// TwinCAT 3 PLC project MC
// ProgramVersion: 3.1.4023.0
// libraries:
//   Tc2_EtherCAT, * (Beckhoff Automation GmbH)
//   Tc2_MC2, * (Beckhoff Automation GmbH)
//   Tc2_MC2_Camming, * (Beckhoff Automation GmbH)
//   Tc2_Standard, * (Beckhoff Automation GmbH)
//   Tc2_System, * (Beckhoff Automation GmbH)
//   Tc3_Module, * (Beckhoff Automation GmbH)
// project tree:
//   / GlobalTextList.TcGTLO, PlcTask.TcTTO, 视图管理器.TcVMO (not stored)
//   POUs/ MAIN.TcPOU, Motion01.TcPOU, Test_SDO.TcPOU
//   VISUs/ hmi.TcVIS
// real-time tasks:
//   TASK PlcTask: cycle T#10ms, priority 20, ADS port 350
//   TASK PlcTask1: cycle T#10ms, priority 21, ADS port 351
// motion (NC):
//   TASK NC-Task 1 SAF: cycle T#2ms, priority 4, ADS port 501
//   TASK NC-Task 1 SVB: cycle T#10ms, priority 8, ADS port 511
//   AXIS Axis 1 (id 1)
//     Dynamic: AccelerationMaximum=30000, DecelerationMaximum=30000, Acceleration=10000, Deceleration=10000, Jerk=5000
//     Velo: Maximum=3300
//     OtherSettings: AllowMotionCmdToSlave=true
//     encoder EncType=1
//       EncPara: ScaleFactorNumerator=60, ScaleFactorDenominator=131072
//         Inc: RefSoftSyncMask=#x0001ffff
//     drive DrvType=5
//       Analog: VeloReferenz=3300, TorqueSetpointScale=10, ScaleFactorActTorque=0.1
//       TimeComp: TaskDelayCycles=1
//     controller CtrType=1
//       CtrPara: PriorControlFactor=1
//         PosDiffControl: Range=100
//         Observer: BandWidth=20
//   AXIS Axis 2 (id 2)
//     OtherSettings: AllowMotionCmdToSlave=true
//     encoder EncType=1
//       EncPara: ScaleFactorNumerator=60, ScaleFactorDenominator=131072
//         Inc: RefSoftSyncMask=#x0001ffff
//     drive DrvType=5
//       Analog: TorqueSetpointScale=10, ScaleFactorActTorque=0.1
//       TimeComp: TaskDelayCycles=1
//     controller CtrType=1
//       CtrPara: PriorControlFactor=1
//         PosDiffControl: Range=100
//         Observer: BandWidth=20
//   AXIS master (id 3)
//     OtherSettings: AllowMotionCmdToSlave=true
//     encoder EncType=19
//       EncPara: ScaleFactorNumerator=60, ScaleFactorDenominator=131072, MaxCount=#xffffffff
//         Inc: RefSoftSyncMask=#x0001ffff
//     drive DrvType=16
//       DrvPara: MaxCount=#xffffffff, DriveControlDWord=#x00020100
//         Analog: TorqueSetpointScale=10, ScaleFactorActTorque=0.1
//         TimeComp: TaskDelayCycles=1
//     controller CtrType=1
//       CtrPara: PriorControlFactor=1
//         PosDiffControl: Range=100
//         Observer: BandWidth=20
//   AXIS slave (id 4)
//     OtherSettings: AllowMotionCmdToSlave=true
//     encoder EncType=19
//       EncPara: ScaleFactorNumerator=60, ScaleFactorDenominator=131072, MaxCount=#xffffffff
//         Inc: RefSoftSyncMask=#x0001ffff
//     drive DrvType=16
//       DrvPara: MaxCount=#xffffffff, DriveControlDWord=#x00020000
//         Analog: TorqueSetpointScale=10, ScaleFactorActTorque=0.1
//         TimeComp: TaskDelayCycles=1
//     controller CtrType=1
//       CtrPara: PriorControlFactor=1
//         PosDiffControl: Range=100
//         Observer: BandWidth=20
// I/O:
//   DEVICE Device 1 (EtherCAT), AmsNetId 5.112.215.215.2.1
//     Term 1 (EK1200) [EK1200-5000 EtherCAT Power supply (2A E-Bus)]
//       Term 2 (EK1110) [EK1110 EtherCAT extension]
//     Drive 3 (ID600E CoE Drive) [ID600E EtherCAT(CoE) Drive]
//     Drive 4 (ID600E CoE Drive) [ID600E EtherCAT(CoE) Drive]
// variable links:
//   NC-Task 1 SAF/Axes/master <-> Device 1 (EtherCAT)/Drive 3 (ID600E CoE Drive)
//     Drive/Inputs/In/nDataIn1 <-> 1st Transmit PDO mapping/Following Error Actual Value
//     Drive/Inputs/In/nDataIn3[0] <-> 1st Transmit PDO mapping/Torque Actual Value
//     Drive/Inputs/In/nDcOutputTime <-> InfoData/DcOutputShift
//     Drive/Inputs/In/nState1 <-> 1st Transmit PDO mapping/Statusword
//     Drive/Inputs/In/nState2 <-> 1st Transmit PDO mapping/Statusword @bit 8
//     Drive/Inputs/In/nState4 @bit 1 <-> WcState/InputToggle
//     Drive/Inputs/In/nState4 <-> WcState/WcState
//     Drive/Inputs/In/nState5 <-> 1st Transmit PDO mapping/Mode of Operation Display
//     Drive/Outputs/Out/nCtrl1 <-> 1st Receive PDO mapping/Controlword
//     Drive/Outputs/Out/nCtrl2 <-> 1st Receive PDO mapping/Controlword @bit 8
//     Drive/Outputs/Out/nCtrl5 <-> 1st Receive PDO mapping/Mode of Operation
//     Drive/Outputs/Out/nDataOut1 <-> 1st Receive PDO mapping/Target Position
//     Drive/Outputs/Out/nDataOut2 <-> 1st Receive PDO mapping/Target Velocity
//     Drive/Outputs/Out/nDataOut4[0] <-> 1st Receive PDO mapping/Target Torque
//     Enc/Inputs/In/nDataIn1 <-> 1st Transmit PDO mapping/Position Actual Value
//     Enc/Inputs/In/nDataIn3 <-> 1st Transmit PDO mapping/Touch Probe 1 Positive Edge Position Value
//     Enc/Inputs/In/nDcInputTime <-> InfoData/DcInputShift
//     Enc/Inputs/In/nState4 @bit 1 <-> WcState/InputToggle
//     Enc/Inputs/In/nState4 <-> WcState/WcState
//     Enc/Outputs/Out/nCtrl5 <-> 1st Receive PDO mapping/Touch Probe Function
//     Enc/Outputs/Out/nCtrl6 <-> 1st Receive PDO mapping/Touch Probe Function @bit 8
//   NC-Task 1 SAF/Axes/slave <-> Device 1 (EtherCAT)/Drive 4 (ID600E CoE Drive)
//     Drive/Inputs/In/nDcOutputTime <-> InfoData/DcOutputShift
//     Drive/Inputs/In/nState1 <-> 2nd Transmit PDO mapping/Statusword
//     Drive/Inputs/In/nState2 <-> 2nd Transmit PDO mapping/Statusword @bit 8
//     Drive/Inputs/In/nState4 @bit 1 <-> WcState/InputToggle
//     Drive/Inputs/In/nState4 <-> WcState/WcState
//     Drive/Outputs/Out/nCtrl1 <-> 2nd Receive PDO mapping/Controlword
//     Drive/Outputs/Out/nCtrl2 <-> 2nd Receive PDO mapping/Controlword @bit 8
//     Drive/Outputs/Out/nDataOut1 <-> 2nd Receive PDO mapping/Target Position
//     Enc/Inputs/In/nDataIn1 <-> 2nd Transmit PDO mapping/Position Actual Value
//     Enc/Inputs/In/nDcInputTime <-> InfoData/DcInputShift
//     Enc/Inputs/In/nState4 @bit 1 <-> WcState/InputToggle
//     Enc/Inputs/In/nState4 <-> WcState/WcState
//   MC/MC Instance <-> NC-Task 1 SAF/Axes/Axis 1
//     PlcTask Inputs/Motion01.Axis01.NcToPlc <-> Outputs/ToPlc
//     PlcTask Outputs/Motion01.Axis01.PlcToNc <-> Inputs/FromPlc
//   MC/MC Instance <-> NC-Task 1 SAF/Axes/Axis 2
//     PlcTask Inputs/Motion01.Axis02.NcToPlc <-> Outputs/ToPlc
//     PlcTask Outputs/Motion01.Axis02.PlcToNc <-> Inputs/FromPlc
//   cam/cam Instance <-> NC-Task 1 SAF/Axes/master
//     PlcTask Inputs/MAIN.master.NcToPlc <-> Outputs/ToPlc
//     PlcTask Outputs/MAIN.master.PlcToNc <-> Inputs/FromPlc
//   cam/cam Instance <-> NC-Task 1 SAF/Axes/slave
//     PlcTask Inputs/MAIN.slave.NcToPlc <-> Outputs/ToPlc
//     PlcTask Outputs/MAIN.slave.PlcToNc <-> Inputs/FromPlc

CONFIGURATION MC
    RESOURCE PLC ON TwinCAT3
        TASK PlcTask(INTERVAL := T#10ms, PRIORITY := 20);
        PROGRAM MAIN WITH PlcTask : MAIN;
    END_RESOURCE
END_CONFIGURATION

// ---- POUs/MAIN.TcPOU
PROGRAM MAIN
VAR
END_VAR

Motion01();
Test_SDO();

END_PROGRAM

// ---- POUs/Motion01.TcPOU
PROGRAM Motion01
VAR
	MC_Power_0				: MC_Power;
	Axis01					: AXIS_REF;
	A1_En					: BOOL;
	MC_Power_1				: MC_Power;
	Axis02					: AXIS_REF;
	A2_En					: BOOL;
	MC_MoveVelocity_0		: MC_MoveVelocity;
	MC_MoveVelocity_1		: MC_MoveVelocity;
	V1_En					: BOOL;
	V2_En					: BOOL;
	MC_Stop_0				: MC_Stop;
	V1_Stp					: BOOL;
	MC_Stop_1				: MC_Stop;
	V2_Stp					: BOOL;
	V1						: LREAL;
	V2						: LREAL;
	MC_Jog_0				: MC_Jog;
	Jog_For					: BOOL;
	MC_MoveRelative_0		: MC_MoveRelative;
	Move_Do					: BOOL;
	MC_SetPosition_0		: MC_SetPosition;
	Set_Do					: BOOL;
	Power_Do				: BOOL;
	MC_Jog_1				: MC_Jog;
	MC_MoveRelative_1		: MC_MoveRelative;
	MC_SetPosition_1		: MC_SetPosition;
	Stop_Do					: BOOL;
	MC_Reset_0				: MC_Reset;
	Reset_Do				: BOOL;
	MC_Reset_1				: MC_Reset;
	MC_GearIn_0				: MC_GearIn;
	MC_GearOut_0			: MC_GearOut;
	Gearin_Do				: BOOL;
	Gearout_Do				: BOOL;
	MC_Home_0				: MC_Home;
	Home_Do					: BOOL;
	Sensor					: BOOL;
	MC_CamIn_0				: MC_CamIn;
	Cam_Do					: BOOL;
	MC_CamOut_0				: MC_CamOut;
	Camout_Do				: BOOL;
END_VAR

MC_Power_0(Axis := Axis01, Enable := Power_Do, Enable_Positive := Power_Do, Enable_Negative := Power_Do); // MC_Power
MC_MoveVelocity_0(
    Axis := Axis01,
    Execute := V1_En,
    Velocity := V1,
    Acceleration := 5000,
    Deceleration := 5000); // MC_MoveVelocity
MC_Stop_0(Axis := Axis01, Execute := Stop_Do, Deceleration := 5000); // MC_Stop
MC_Power_1(Axis := Axis02, Enable := Power_Do, Enable_Positive := Power_Do, Enable_Negative := Power_Do); // MC_Power
MC_MoveVelocity_1(
    Axis := Axis02,
    Execute := V2_En,
    Velocity := V2,
    Acceleration := 5000,
    Deceleration := 5000); // MC_MoveVelocity
MC_Stop_1(Axis := Axis02, Execute := Stop_Do, Deceleration := 5000); // MC_Stop
MC_Jog_0(Axis := Axis01, JogForward := Jog_For); // MC_Jog
MC_MoveRelative_0(Axis := Axis01, Execute := Move_Do, Distance := 1000, Velocity := 100); // MC_MoveRelative
MC_SetPosition_0(Axis := Axis01, Execute := Set_Do, Position := 0); // MC_SetPosition
MC_Jog_1(Axis := Axis02); // MC_Jog
MC_MoveRelative_1(Axis := Axis02, Execute := Move_Do); // MC_MoveRelative
MC_SetPosition_1(Axis := Axis02, Execute := Set_Do, Position := 0); // MC_SetPosition
MC_Reset_0(Axis := Axis01, Execute := Reset_Do); // MC_Reset
MC_Reset_1(Axis := Axis02, Execute := Reset_Do); // MC_Reset
MC_GearIn_0(
    Master := Axis01,
    Slave := Axis02,
    Execute := Gearin_Do,
    RatioNumerator := 1,
    RatioDenominator := 2); // MC_GearIn
MC_GearOut_0(Slave := Axis02, Execute := Gearout_Do); // MC_GearOut
MC_Home_0(Axis := Axis01, Execute := Home_Do, Position := 0, bCalibrationCam := Sensor); // MC_Home
MC_CamIn_0(Master := Axis01, Slave := Axis02, Execute := Cam_Do, CamTableID := 1); // MC_CamIn
MC_CamOut_0(Slave := Axis02, Execute := Camout_Do); // MC_CamOut

END_PROGRAM

// ---- POUs/Test_SDO.TcPOU
PROGRAM Test_SDO
VAR
	fbSdoRead  : FB_EcCoESdoRead;
    sNetId     : T_AmsNetId := '5.112.215.215.2.1';
    bExecute   : BOOL;
    nSlaveAddr : UINT := 1002;
    nIndex     : WORD := 16#4106;
    nSubIndex  : BYTE :=0;
    vendorId   : UDINT;
    bError     : BOOL;
    nErrId     : UDINT;
	
	fbSdoWrite 	: FB_EcCoESdoWrite;
    sNetId1     : T_AmsNetId := '5.112.215.215.2.1'; (* NetId of EtherCAT Master *)
    nSlaveAddr1 : UINT := 1002; (* Port Number of EtherCAT Slave *)
    nIndex1     : WORD := 16#5F04; (* CoE Object Index *)
    nSubIndex1  : BYTE := 0; (* Subindex of CoE Object *)
    nValue1     : UINT := 0; (* variable to be written to the CoE Object *)(*1为编码器报警清除，2为编码器圈数清零*)
    bExecute1   : BOOL; (* rising edge starts writing to the CoE Object *)
    bError1     : BOOL;
    nErrId1     : UDINT;
END_VAR

fbSdoRead(
	sNetId:= sNetId,
	nSlaveAddr :=nSlaveAddr, 
	nIndex:=nIndex, 
	nSubIndex :=nSubIndex, 
	pDstBuf:= ADR(vendorId), 
	cbBufLen:=SIZEOF(vendorId),
	bExecute:=bExecute
);

bError:=fbSdoRead.bError;
nErrId:=fbSdoRead.nErrId;

fbSdoWrite(
    sNetId     := sNetId1,
    nSlaveAddr := nSlaveAddr1,
    nIndex     := nIndex1,
    nSubIndex  := nSubIndex1,
    pSrcBuf    := ADR(nValue1),
    cbBufLen   := SIZEOF(nValue1),
    bExecute   := bExecute1
);

END_PROGRAM

// ---- GlobalTextList.TcGTLO
TEXTLIST GlobalTextList
  635 = 'Axis1:%.2f'
  633 = 'Axis2:%.2f'
  414 = '使能'
  855 = '停止'
  600 = '凸轮耦合'
  371 = '凸轮解耦'
  444 = '原点信号'
  861 = '回原点'
  119 = '复位'
  925 = '点动'
  753 = '电子齿轮'
  227 = '设置零点'
  478 = '走增量位置'
  521 = '轴1使能'
  672 = '轴1点动'
  972 = '齿轮解耦'
END_TEXTLIST

// ---- VISUs/hmi.TcVIS
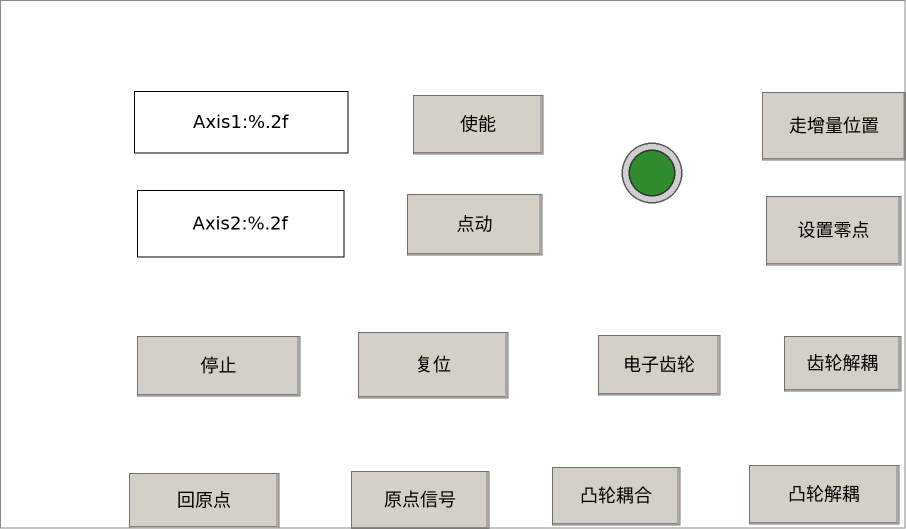
VISUALIZATION hmi  // 906x529
    Rectangle (134,91 214x62), "Axis1:%.2f", text variable: Motion01.Axis01.NcToPlc.ActPos
    Rectangle (137,190 207x67), "Axis2:%.2f", text variable: Motion01.Axis02.NcToPlc.ActPos
    Button (413,95 130x59), "使能"
        toggle Motion01.Power_Do
    Button (407,194 135x61), "点动"
        toggle Motion01.Jog_For
    Lamp1 (617,138 70x70), variable: Motion01.Axis01.NcToPlc.StateDWord.20, style: Lamp-Lamp1-Green
    Button (762,92 144x68), "走增量位置"
        tap Motion01.Move_Do
    Button (766,196 135x69), "设置零点"
        tap Motion01.Set_Do
    Button (137,336 163x60), "停止"
        tap Motion01.Stop_Do
    Button (358,332 150x66), "复位"
        tap Motion01.Reset_Do
    Button (598,335 122x60), "电子齿轮"
        tap Motion01.Gearin_Do
    Button (784,336 117x55), "齿轮解耦"
        tap Motion01.Gearout_Do
    Button (129,473 150x55), "回原点"
        tap Motion01.Home_Do
    Button (351,471 138x58), "原点信号"
        tap Motion01.Sensor
    Button (552,467 128x58), "凸轮耦合"
        tap Motion01.Cam_Do
    Button (749,465 150x59), "凸轮解耦"
        tap Motion01.Camout_Do
END_VISUALIZATION
